{attribute addProperty BoxType "ELM3102-0000-0016"}
{attribute addProperty Id "PAI_Status_Channel_1AT %I*PAI_Status_Channel_CF7232B03240PAI_Samples_1_Channel_1AT %I*PAI_Samples_1_Channel_4FE6FA0C3240PAI_Timestamp_Channel_1AT %I*PAI_Timestamp_Channel_54B31DA16480PAI_Status_Channel_2AT %I*PAI_Status_Channel_CF7232B03240PAI_Samples_1_Channel_2AT %I*PAI_Samples_1_Channel_4FE6FA0C3240WcStateAT %I*WcState_F855686C1620InfoDataAT %I*InfoData_0BDED7BF144180"}
{attribute addProperty CRC "3627193320"}
{attribute addProperty SizeInBites "352"}
{attribute addProperty SizeInBytes "44"}
TYPE ELM3102_1C598C25 :
STRUCT
	{attribute addProperty Name "PAI_Status_Channel_1"}
	PAI_Status_Channel_1 : PAI_Status_Channel_CF7232B0;
	{attribute addProperty Name "PAI_Samples_1_Channel_1"}
	PAI_Samples_1_Channel_1 : PAI_Samples_1_Channel_4FE6FA0C;
	{attribute addProperty Name "PAI_Timestamp_Channel_1"}
	PAI_Timestamp_Channel_1 : PAI_Timestamp_Channel_54B31DA1;
	{attribute addProperty Name "PAI_Status_Channel_2"}
	PAI_Status_Channel_2 : PAI_Status_Channel_CF7232B0;
	{attribute addProperty Name "PAI_Samples_1_Channel_2"}
	PAI_Samples_1_Channel_2 : PAI_Samples_1_Channel_4FE6FA0C;
	{attribute addProperty Name "WcState"}
	WcState : WcState_F855686C;
	{attribute addProperty Name "InfoData"}
	InfoData : InfoData_0BDED7BF;
END_STRUCT
END_TYPE

(* stored: Version 1.2.0.0, ProductVersion 3.1.4024.9
   DUT ELM3102_1C598C25: Id {64290897-8b4e-434d-824f-d88e2f3d3720} *)
